// SIMATIC S7-200 SMART project (STEP 7-Micro/WIN SMART), CPU SR20

SYMBOL_TABLE 系统符号
Always_On        SM0.0    // 始终接通
Clock_1s         SM0.5    // 针对 1 s 的周期时间，时钟脉冲接通 0.5 s，断开 0.5 s.
END_SYMBOL_TABLE

SYMBOL_TABLE Modbus TCP Server (v1.0)
mMsgBuf_Length   VW200    // Offset: 4
END_SYMBOL_TABLE

ORGANIZATION_BLOCK 程序块:OB1
TITLE=程序注释
BEGIN
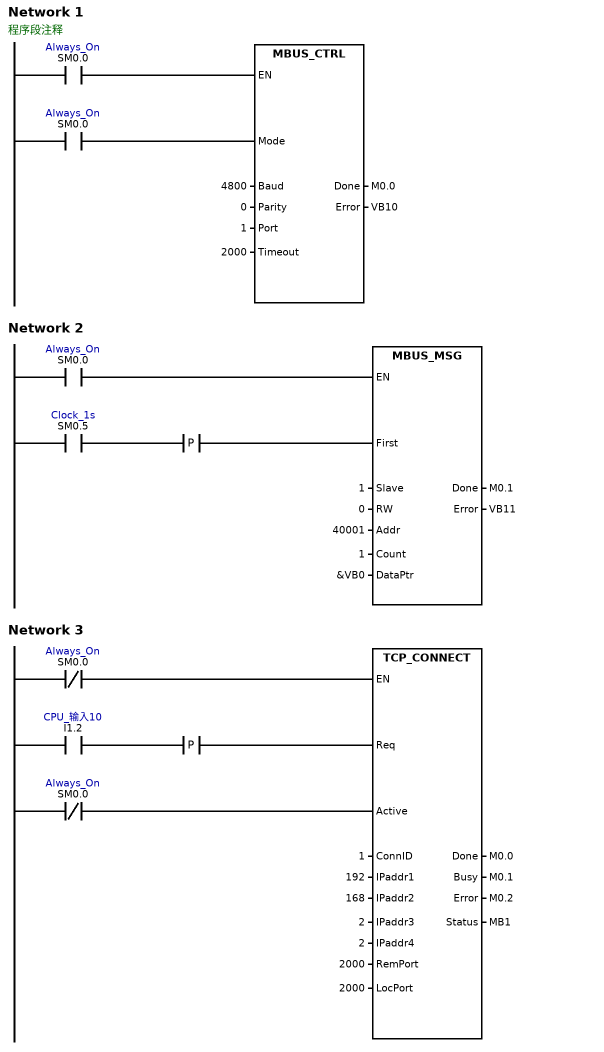
Network 1
// 程序段注释
LD     Always_On:SM0.0
=      L60.0
LD     Always_On:SM0.0
=      L63.7
LD     L60.0
CALL   MBUS_CTRL:SBR2, L63.7, 4800, 0, 1, 2000, M0.0, VB10
Network 2
LD     Always_On:SM0.0
=      L60.0
LD     Clock_1s:SM0.5
EU
=      L63.7
LD     L60.0
CALL   MBUS_MSG:SBR3, L63.7, 1, 0, 40001, 1, &VB0, M0.1, VB11
Network 3
LDN    Always_On:SM0.0
=      L60.0
LD     CPU_输入10:I1.2
EU
=      L63.7
LDN    Always_On:SM0.0
=      L63.6
LD     L60.0
CALL   TCP_CONNECT:SBR6, L63.7, L63.6, 1, 192, 168, 2, 2, 2000, 2000, M0.0, M0.1, M0.2, MB1
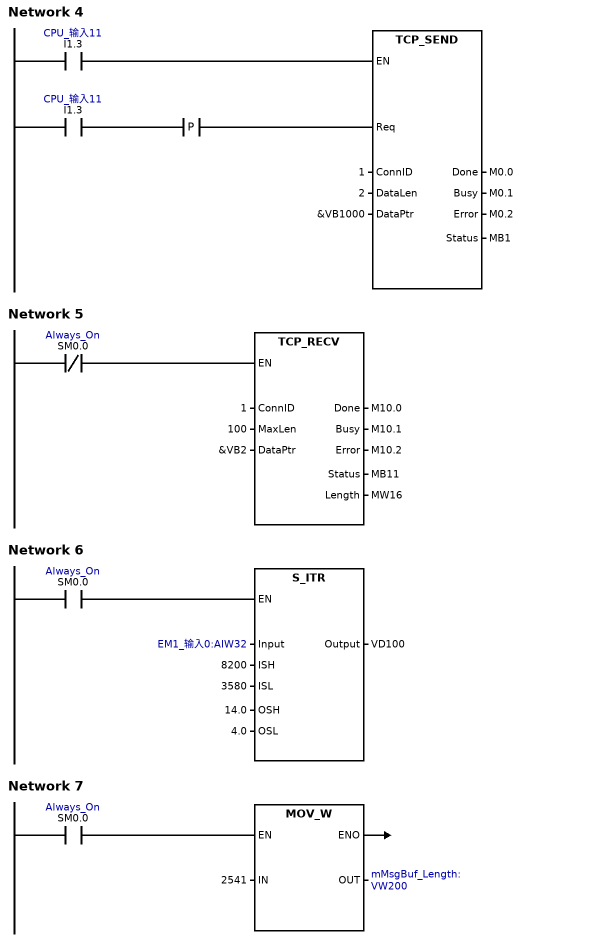
Network 4
LD     CPU_输入11:I1.3
=      L60.0
LD     CPU_输入11:I1.3
EU
=      L63.7
LD     L60.0
CALL   TCP_SEND:SBR7, L63.7, 1, 2, &VB1000, M0.0, M0.1, M0.2, MB1
Network 5
LDN    Always_On:SM0.0
CALL   TCP_RECV:SBR9, 1, 100, &VB2, M10.0, M10.1, M10.2, MB11, MW16
Network 6
LD     Always_On:SM0.0
CALL   S_ITR:SBR13, EM1_输入0:AIW32, 8200, 3580, 14.0, 4.0, VD100
Network 7
LD     Always_On:SM0.0
MOVW   2541, mMsgBuf_Length:VW200
END_ORGANIZATION_BLOCK

// SBR1: protected block, not included

// SBR2: protected block, not included

// SBR3: protected block, not included

// SBR4: protected block, not included

// SBR5: protected block, not included

// SBR6: protected block, not included

// SBR7: protected block, not included

// SBR9: protected block, not included

// SBR10: protected block, not included

// SBR11: protected block, not included

// SBR12: protected block, not included

// SBR13: protected block, not included
